(* What operations should be used to compare gauge status *)
TYPE ST_SBGaugeReadingsOp :
STRUCT
	eDPPiraniOp : E_GaugeCompOp; // LXLHN:GPI:03
	eDPColdCathodeOp : E_GaugeCompOp; // LXLHN:GCC:02
	ePumpStationPirani1Op : E_GaugeCompOp; // LXLHN:GPI:01
	ePumpStationPirani2Op : E_GaugeCompOp; // LXLHN:GPI:02
	ePumpStationColdCathodeOp : E_GaugeCompOp; // LXLHN:GCC:01
END_STRUCT
END_TYPE

(* stored: Version 1.1.0.1, ProductVersion 3.1.4022.18
   DUT ST_SBGaugeReadingsOp: Id {ebf512b5-0f6b-409e-b8c4-a238edda22c0} *)
